// SIMATIC S7-200 project (STEP 7-Micro/WIN), CPU 221 REL 01.10

ORGANIZATION_BLOCK 主程序:OB1
TITLE=程序注释
BEGIN
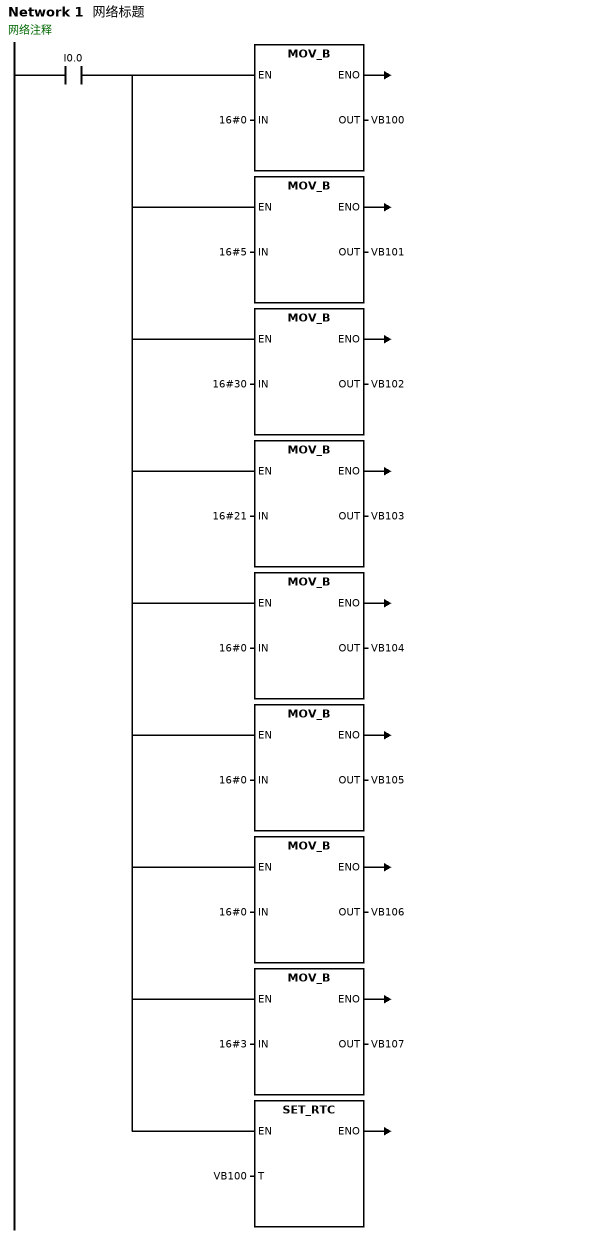
Network 1 // 网络标题
// 网络注释
LD     I0.0
MOVB   16#0, VB100
MOVB   16#5, VB101
MOVB   16#30, VB102
MOVB   16#21, VB103
MOVB   16#0, VB104
MOVB   16#0, VB105
MOVB   16#0, VB106
MOVB   16#3, VB107
TODW   VB100
END_ORGANIZATION_BLOCK
